FUNCTION_BLOCK ST80a
VAR
	_promenlivaIvana	: BOOL;
	_test : BOOL;
	_ivana : BOOL; 
END_VAR

METHOD PROTECTED _Ready 
VAR_INPUT
END_VAR
_test:= TRUE; 
_promenlivaIvana:= TRUE;
END_METHOD

END_FUNCTION_BLOCK

(* stored: Version 1.1.0.1, ProductVersion 3.1.4024.12
   POU ST80a: Id {ebc57cc3-e53c-4a10-a66c-718a2d623872}, SpecialFunc None
   Method _Ready: Id {1c117af2-23f0-45c4-ae45-7896f814997b} *)
